// Mitsubishi GX Works2 project: GROUP34   PLC: FX3G

// global labels: Global1
VAR_GLOBAL
  Start_day_button AT X007 : BOOL;
  Insert_stock_once AT M9 : BOOL;
  Petel_input AT D1100 : REAL;
  Petel_stock AT D1102 : REAL;
  Lemon_input AT D1104 : REAL;
  Lemon_stock AT D1106 : REAL;
  Stabilizer_input AT D1108 : REAL;
  Stabilizer_stock AT D1110 : REAL;
  Gummy_input AT D1112 : REAL;
  Gummy_stock AT D1114 : REAL;
  Out_of_stock_reg AT M13 : BOOL;
  Emergency_button AT X005 : BOOL;
  End_day AT M1 : BOOL;
  Start_production AT M2 : BOOL;
  Start_packing AT X004 : BOOL;
  Choose_type AT X001 : BOOL;
END_VAR
VAR_GLOBAL CONSTANT
  Min_petel : REAL := 280;
  Min_lemon : REAL := 455;
  Min_stabilazer : REAL := 105;
  Min_gummy : REAL := 28;
  Min_petel_pinuk : REAL := 385;
  Min_lemon_pinuk : REAL := 665;
  Min_stabilazer_pinuk : REAL := 210;
  Min_gummy_pinuk : REAL := 70;
END_VAR
VAR_GLOBAL
  Out_of_stock_pinuk AT M14 : BOOL;
  Start_day_bulb AT Y007 : BOOL;
  Analog_output AT D8282 : INT;
  Tot_storage AT D1128 : REAL;
END_VAR
VAR_GLOBAL CONSTANT
  Div_analog1 : REAL := 400;
END_VAR
VAR_GLOBAL
  Start_preperation AT M6 : BOOL;
END_VAR
VAR_GLOBAL CONSTANT
  Choose_reg : REAL := 5;
END_VAR
VAR_GLOBAL
  Make_reg AT M7 : BOOL;
  Make_pinuk AT M8 : BOOL;
  Div_output AT D1170 : REAL;
  Is_mix AT TC1 : BOOL;
END_VAR
VAR_GLOBAL CONSTANT
  Wait_5_sec : INT := 50;
END_VAR
VAR_GLOBAL
  Preperation_lamp AT Y000 : BOOL;
  Ice_cream_reg_stage AT M17 : BOOL;
  Ice_cream_pinuk_stage AT M18 : BOOL;
  Petel_preperation AT D1118 : REAL;
END_VAR
VAR_GLOBAL CONSTANT
  Weight_reg_petel_ice_cream : REAL := 350;
END_VAR
VAR_GLOBAL
  Lemon_preperation AT D1120 : REAL;
END_VAR
VAR_GLOBAL CONSTANT
  Weight_reg_lemon_ice_cream : REAL := 490;
  Weight_pinuk_petel_ice_cream : REAL := 560;
  Weight_pinuk_lemon_ice_cream : REAL := 700;
END_VAR
VAR_GLOBAL
  Start_cooling AT X002 : BOOL;
  Cool_petel AT D1122 : REAL;
  Cooling AT M22 : BOOL;
  Is_cooling AT TC2 : BOOL;
END_VAR
VAR_GLOBAL CONSTANT
  Cooling_time : INT := 80;
END_VAR
VAR_GLOBAL
  Cooling_lamp AT M26 : BOOL;
  Temp_sensor_upper10 AT X003 : BOOL;
  Finish_mix AT TS1 : BOOL;
  Finish_cooling AT TS2 : BOOL;
  Cooling_finish AT TS2 : BOOL;
  Cooling_inprocess AT M21 : BOOL;
  Temp_under10 AT M23 : BOOL;
  Cool_lemon AT D1124 : REAL;
  Mix_Tot AT D1126 : REAL;
  Finish_move_icecream AT M25 : BOOL;
END_VAR
VAR_GLOBAL CONSTANT
  Gummy_reg : REAL := 28;
END_VAR
VAR_GLOBAL
  Finish_move AT M24 : BOOL;
END_VAR
VAR_GLOBAL CONSTANT
  Gummy_pinuk : REAL := 70;
END_VAR
VAR_GLOBAL
  Finish_mix_pinuk AT M12 : BOOL;
  Help_Blinking AT M0 : BOOL;
  Blink_y5 AT TC3 : BOOL;
END_VAR
VAR_GLOBAL CONSTANT
  Counter_blink_y5 : INT := 5;
END_VAR
VAR_GLOBAL
  Stop_blink_y5 AT TS3 : BOOL;
  Y5_bulb AT Y005 : BOOL;
  Finish_mix_reg AT M11 : BOOL;
  Blink_y6 AT TC4 : BOOL;
END_VAR
VAR_GLOBAL CONSTANT
  Counter_blink_y6 : INT := 5;
END_VAR
VAR_GLOBAL
  Stop_blink_y6 AT TS4 : BOOL;
  Y6_bulb AT Y006 : BOOL;
  Timer_blinking_reg AT TC5 : BOOL;
END_VAR
VAR_GLOBAL CONSTANT
  Counter_3sec : INT := 30;
END_VAR
VAR_GLOBAL
  Stop_reg_mix AT TS5 : BOOL;
  Timer_blinking_pinuk AT TC6 : BOOL;
END_VAR
VAR_GLOBAL CONSTANT
  Counter_5sec : INT := 50;
END_VAR
VAR_GLOBAL
  Stop_pinuk_mix AT TS6 : BOOL;
  Save_type AT D1200 : REAL;
  Test AT D1500 : REAL;
  Analog_to_real AT D6000 : REAL;
  Insert_to_storage AT X000 : BOOL;
END_VAR
VAR_GLOBAL CONSTANT
  Counter_7 : INT := 7;
END_VAR
VAR_GLOBAL
  Count_in_storage AT CC1 : BOOL;
  Stocking_bulb AT M27 : BOOL;
  finish_stocking AT CS1 : BOOL;
END_VAR
VAR_GLOBAL CONSTANT
  Add_1 : REAL := 1.0;
  Div_analog2 : REAL := 40.0;
END_VAR
VAR_GLOBAL
  num_of_packs AT D1130 : REAL;
  Analog_input1 AT D8280 : INT;
  Cooling_stocking_lamp AT Y002 : BOOL;
  Is_out_of_stock AT M29 : BOOL;
  Finish_cool AT M26 : BOOL;
END_VAR

// task Task_01 (event TRUE, interval 0, priority 31): POU_01

PROGRAM POU_01
(* structured ladder/FBD written out as ST: instructions are called as NAME(EN, inputs, outputs); _pN, _eN, _tN stand for wires *)
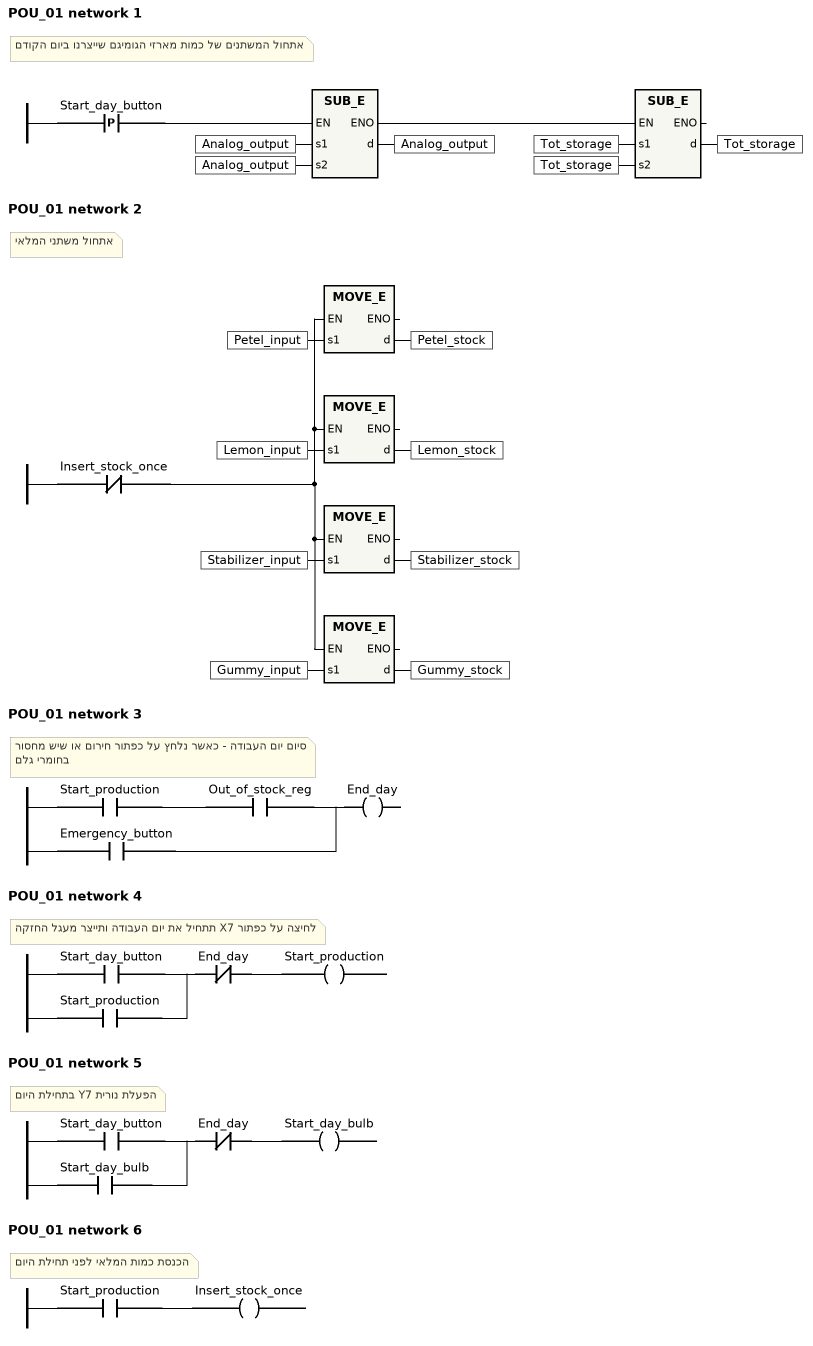
(* network 1 *)
(* אתחול המשתנים של כמות מארזי הגומיגם שייצרנו ביום הקודם *)
_e1 := SUB_E(LDP(TRUE, Start_day_button), Analog_output, Analog_output, Analog_output);
SUB_E(_e1, Tot_storage, Tot_storage, Tot_storage);
(* network 2 *)
(* אתחול משתני המלאי *)
_p1 := NOT Insert_stock_once;
MOVE_E(_p1, Petel_input, Petel_stock);
MOVE_E(_p1, Lemon_input, Lemon_stock);
MOVE_E(_p1, Stabilizer_input, Stabilizer_stock);
MOVE_E(_p1, Gummy_input, Gummy_stock);
(* network 3 *)
(* סיום יום העבודה - כאשר נלחץ על כפתור חירום או שיש מחסור בחומרי גלם *)
End_day := (Start_production AND Out_of_stock_reg) OR Emergency_button;
(* network 4 *)
(* לחיצה על כפתור X7 תתחיל את יום העבודה ותייצר מעגל החזקה *)
Start_production := (Start_day_button OR Start_production) AND NOT End_day;
(* network 5 *)
(* הפעלת נורית Y7 בתחילת היום *)
Start_day_bulb := (Start_day_button OR Start_day_bulb) AND NOT End_day;
(* network 6 *)
(* הכנסת כמות המלאי לפני תחילת היום *)
Insert_stock_once := Start_production;
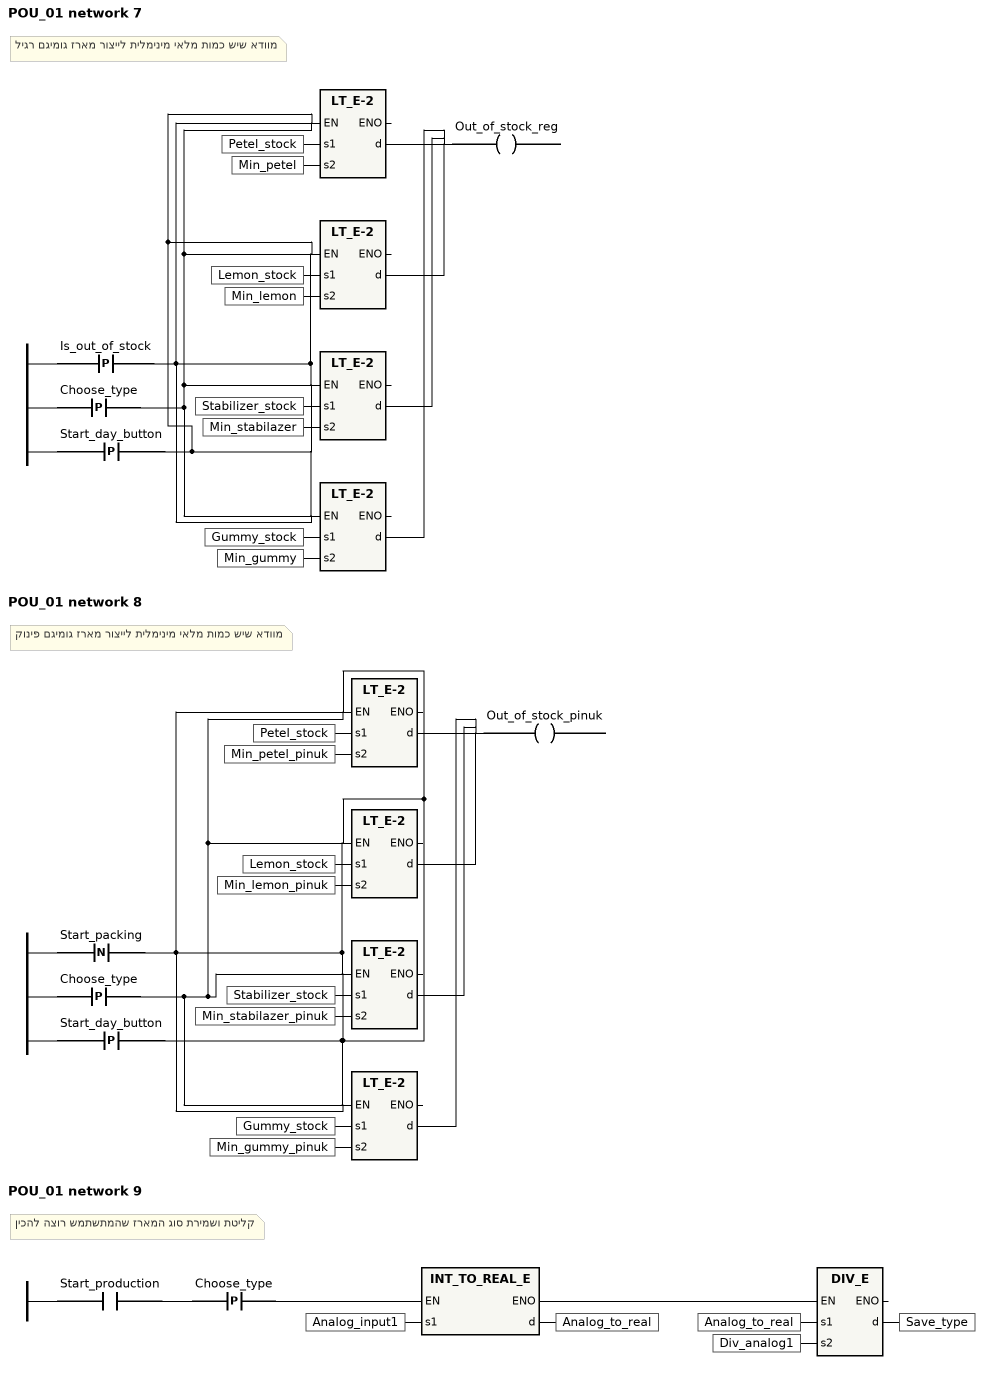
(* network 7 *)
(* מוודא שיש כמות מלאי מינימלית לייצור מארז גומיגם רגיל *)
_p1 := LDP(TRUE, Is_out_of_stock) OR LDP(TRUE, Choose_type) OR LDP(TRUE, Start_day_button);
LT_E(_p1, Petel_stock, Min_petel, _t2);
LT_E(_p1, Lemon_stock, Min_lemon, _t3);
LT_E(_p1, Stabilizer_stock, Min_stabilazer, _t4);
LT_E(_p1, Gummy_stock, Min_gummy, _t5);
Out_of_stock_reg := _t2 OR _t3 OR _t4 OR _t5;
(* network 8 *)
(* מוודא שיש כמות מלאי מינימלית לייצור מארז גומיגם פינוק *)
_p1 := LDF(TRUE, Start_packing) OR LDP(TRUE, Choose_type) OR LDP(TRUE, Start_day_button);
LT_E(_p1, Petel_stock, Min_petel_pinuk, _t2);
LT_E(_p1, Lemon_stock, Min_lemon_pinuk, _t3);
LT_E(_p1, Stabilizer_stock, Min_stabilazer_pinuk, _t4);
LT_E(_p1, Gummy_stock, Min_gummy_pinuk, _t5);
Out_of_stock_pinuk := _t2 OR _t3 OR _t4 OR _t5;
(* network 9 *)
(* קליטת ושמירת סוג המארז שהמתשתמש רוצה להכין *)
_e1 := INT_TO_REAL_E(Start_production AND LDP(TRUE, Choose_type), Analog_input1, Analog_to_real);
DIV_E(_e1, Analog_to_real, Div_analog1, Save_type);
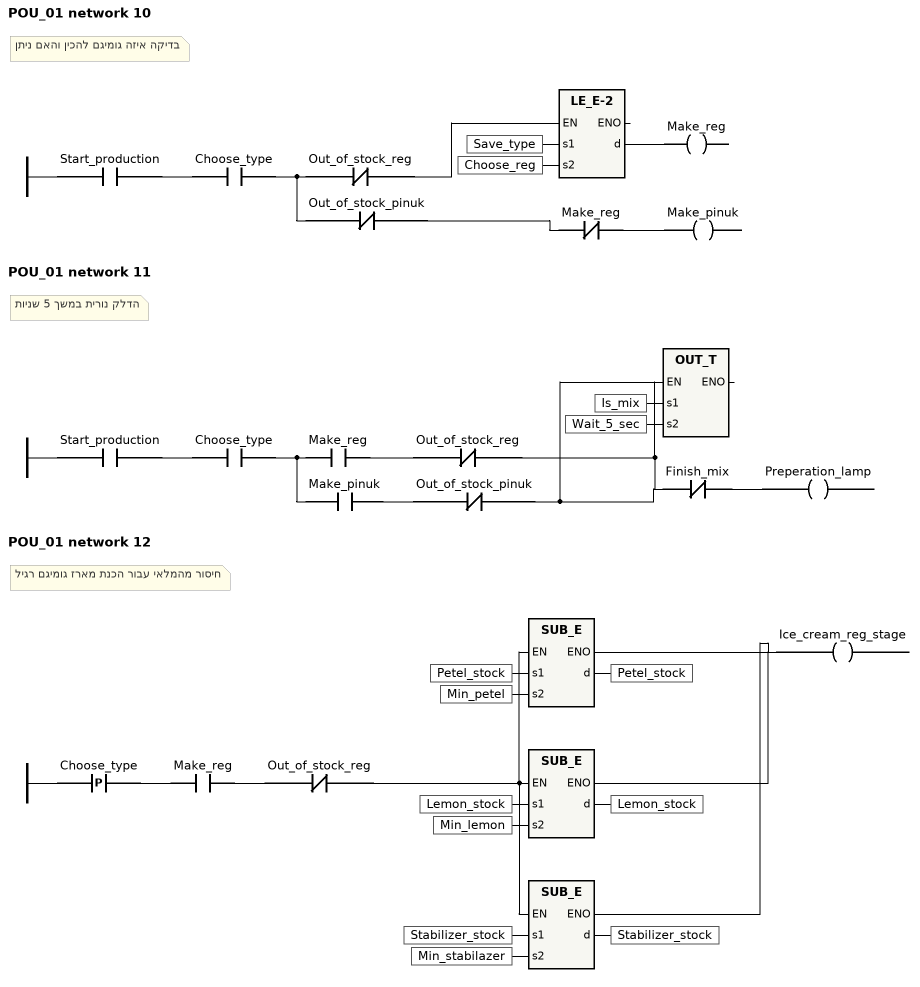
(* network 10 *)
(* בדיקה איזה גומיגם להכין והאם ניתן *)
_p1 := Start_production AND Choose_type;
LE_E(_p1 AND NOT Out_of_stock_reg, Save_type, Choose_reg, _t2);
Make_reg := _t2;
Make_pinuk := _p1 AND NOT Out_of_stock_pinuk AND NOT Make_reg;
(* network 11 *)
(* הדלק נורית במשך 5 שניות *)
_p1 := Start_production AND Choose_type;
_p2 := (_p1 AND Make_reg AND NOT Out_of_stock_reg) OR (_p1 AND Make_pinuk AND NOT Out_of_stock_pinuk);
OUT_T(_p2, Is_mix, Wait_5_sec);
Preperation_lamp := _p2 AND NOT Finish_mix;
(* network 12 *)
(* חיסור מהמלאי עבור הכנת מארז גומיגם רגיל *)
_p1 := LDP(TRUE, Choose_type) AND Make_reg AND NOT Out_of_stock_reg;
_e2 := SUB_E(_p1, Petel_stock, Min_petel, Petel_stock);
_e3 := SUB_E(_p1, Lemon_stock, Min_lemon, Lemon_stock);
_e4 := SUB_E(_p1, Stabilizer_stock, Min_stabilazer, Stabilizer_stock);
Ice_cream_reg_stage := _e2 OR _e3 OR _e4;
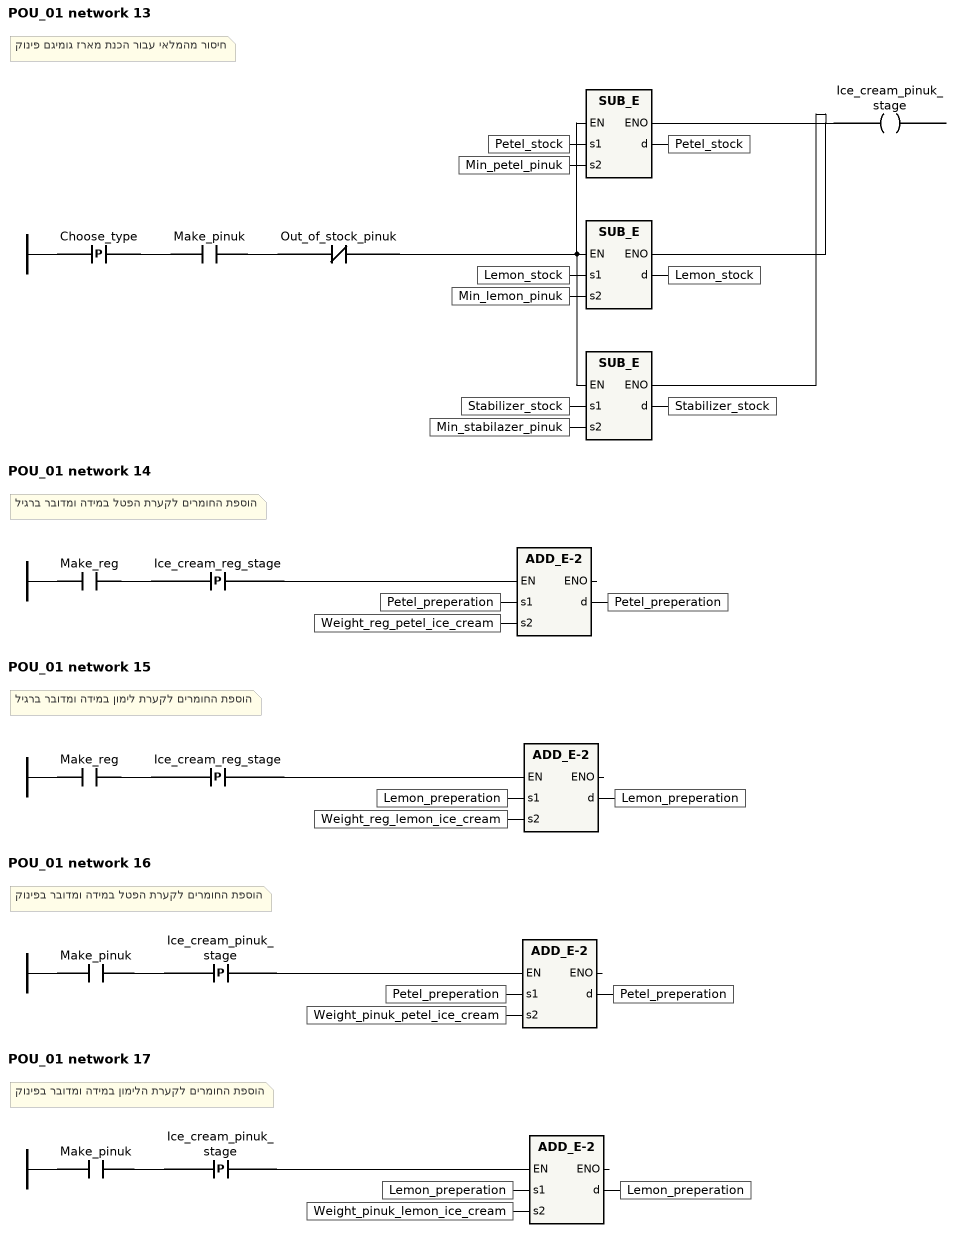
(* network 13 *)
(* חיסור מהמלאי עבור הכנת מארז גומיגם פינוק *)
_p1 := LDP(TRUE, Choose_type) AND Make_pinuk AND NOT Out_of_stock_pinuk;
_e2 := SUB_E(_p1, Petel_stock, Min_petel_pinuk, Petel_stock);
_e3 := SUB_E(_p1, Lemon_stock, Min_lemon_pinuk, Lemon_stock);
_e4 := SUB_E(_p1, Stabilizer_stock, Min_stabilazer_pinuk, Stabilizer_stock);
Ice_cream_pinuk_stage := _e2 OR _e3 OR _e4;
(* network 14 *)
(* הוספת החומרים לקערת הפטל במידה ומדובר ברגיל *)
ADD_E(Make_reg AND LDP(TRUE, Ice_cream_reg_stage), Petel_preperation, Weight_reg_petel_ice_cream, Petel_preperation);
(* network 15 *)
(* הוספת החומרים לקערת לימון במידה ומדובר ברגיל *)
ADD_E(Make_reg AND LDP(TRUE, Ice_cream_reg_stage), Lemon_preperation, Weight_reg_lemon_ice_cream, Lemon_preperation);
(* network 16 *)
(* הוספת החומרים לקערת הפטל במידה ומדובר בפינוק *)
ADD_E(Make_pinuk AND LDP(TRUE, Ice_cream_pinuk_stage), Petel_preperation, Weight_pinuk_petel_ice_cream, Petel_preperation);
(* network 17 *)
(* הוספת החומרים לקערת הלימון במידה ומדובר בפינוק *)
ADD_E(Make_pinuk AND LDP(TRUE, Ice_cream_pinuk_stage), Lemon_preperation, Weight_pinuk_lemon_ice_cream, Lemon_preperation);
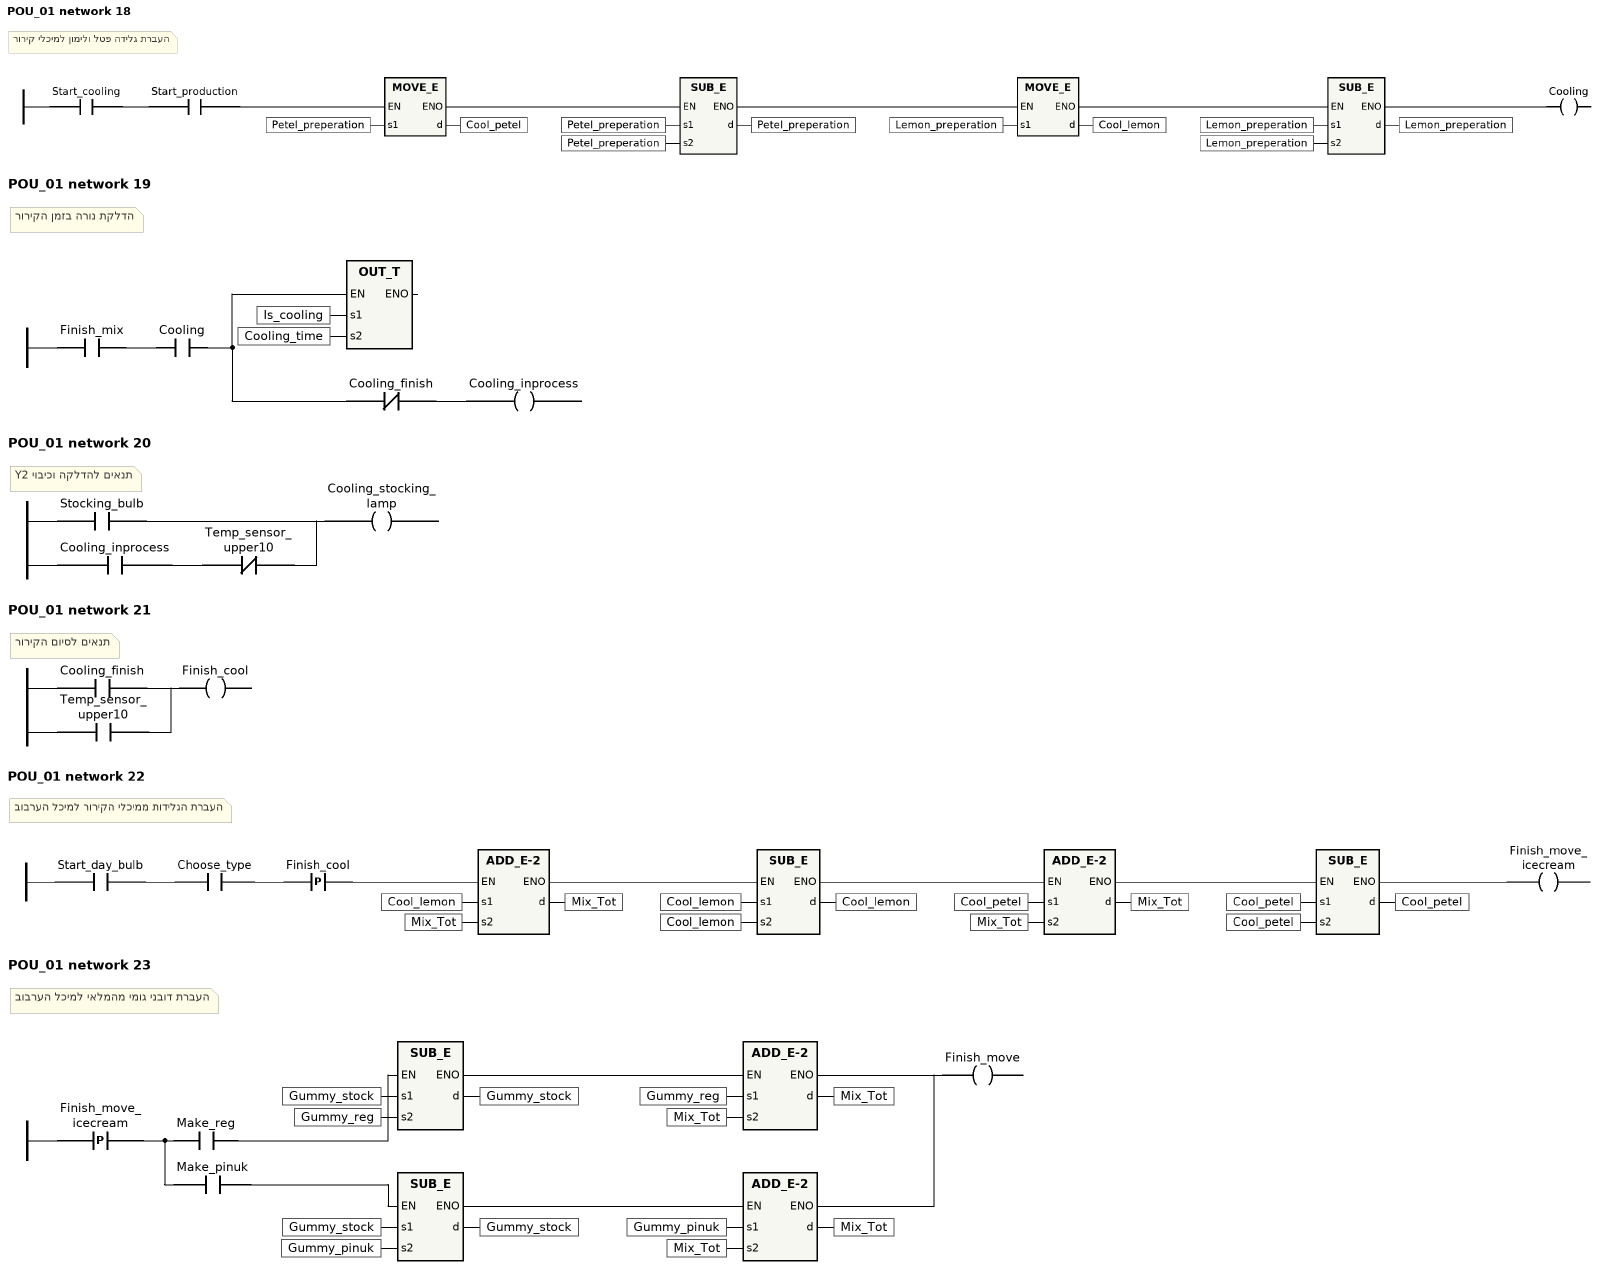
(* network 18 *)
(* העברת גלידה פטל ולימון למיכלי קירור *)
_e1 := MOVE_E(Start_cooling AND Start_production, Petel_preperation, Cool_petel);
_e2 := SUB_E(_e1, Petel_preperation, Petel_preperation, Petel_preperation);
_e3 := MOVE_E(_e2, Lemon_preperation, Cool_lemon);
_e4 := SUB_E(_e3, Lemon_preperation, Lemon_preperation, Lemon_preperation);
Cooling := _e4;
(* network 19 *)
(* הדלקת נורה בזמן הקירור *)
_p1 := Finish_mix AND Cooling;
OUT_T(_p1, Is_cooling, Cooling_time);
Cooling_inprocess := _p1 AND NOT Cooling_finish;
(* network 20 *)
(* תנאים להדלקה וכיבוי Y2 *)
Cooling_stocking_lamp := Stocking_bulb OR (Cooling_inprocess AND NOT Temp_sensor_upper10);
(* network 21 *)
(* תנאים לסיום הקירור *)
Finish_cool := Cooling_finish OR Temp_sensor_upper10;
(* network 22 *)
(* העברת הגלידות ממיכלי הקירור למיכל הערבוב *)
_e1 := ADD_E(Start_day_bulb AND Choose_type AND LDP(TRUE, Finish_cool), Cool_lemon, Mix_Tot, Mix_Tot);
_e2 := SUB_E(_e1, Cool_lemon, Cool_lemon, Cool_lemon);
_e3 := ADD_E(_e2, Cool_petel, Mix_Tot, Mix_Tot);
_e4 := SUB_E(_e3, Cool_petel, Cool_petel, Cool_petel);
Finish_move_icecream := _e4;
(* network 23 *)
(* העברת דובני גומי מהמלאי למיכל הערבוב *)
_p1 := LDP(TRUE, Finish_move_icecream);
_e2 := SUB_E(_p1 AND Make_reg, Gummy_stock, Gummy_reg, Gummy_stock);
_e3 := ADD_E(_e2, Gummy_reg, Mix_Tot, Mix_Tot);
_e4 := SUB_E(_p1 AND Make_pinuk, Gummy_stock, Gummy_pinuk, Gummy_stock);
_e5 := ADD_E(_e4, Gummy_pinuk, Mix_Tot, Mix_Tot);
Finish_move := _e3 OR _e5;
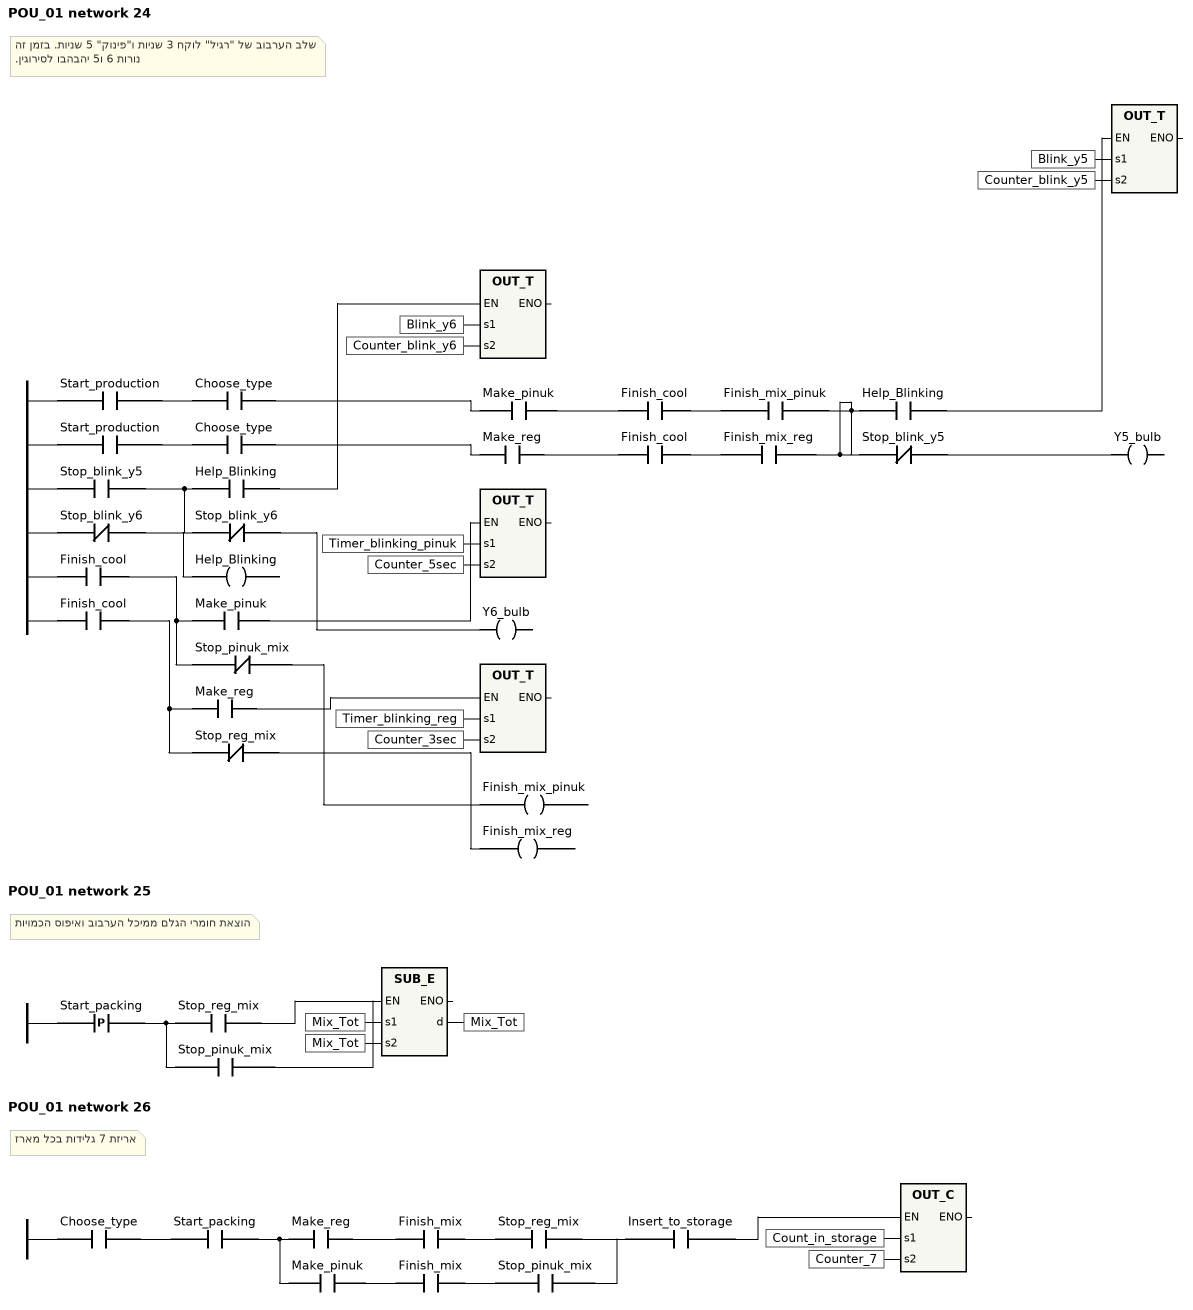
(* network 24 *)
(* שלב הערבוב של "רגיל" לוקח 3 שניות ו"פינוק" 5 שניות. בזמן זה נורות 6 ו5 יהבהבו לסירוגין. *)
_p1 := (Start_production AND Choose_type AND Make_pinuk AND Finish_cool AND Finish_mix_pinuk) OR (Start_production AND Choose_type AND Make_reg AND Finish_cool AND Finish_mix_reg);
OUT_T(_p1 AND Help_Blinking, Blink_y5, Counter_blink_y5);
Y5_bulb := _p1 AND NOT Stop_blink_y5;
OUT_T(Stop_blink_y5 AND Help_Blinking, Blink_y6, Counter_blink_y6);
Y6_bulb := Stop_blink_y5 AND NOT Stop_blink_y6;
Help_Blinking := NOT Stop_blink_y6;
OUT_T(Finish_cool AND Make_pinuk, Timer_blinking_pinuk, Counter_5sec);
Finish_mix_pinuk := Finish_cool AND NOT Stop_pinuk_mix;
OUT_T(Finish_cool AND Make_reg, Timer_blinking_reg, Counter_3sec);
Finish_mix_reg := Finish_cool AND NOT Stop_reg_mix;
(* network 25 *)
(* הוצאת חומרי הגלם ממיכל הערבוב ואיפוס הכמויות *)
_p1 := LDP(TRUE, Start_packing);
SUB_E((_p1 AND Stop_reg_mix) OR (_p1 AND Stop_pinuk_mix), Mix_Tot, Mix_Tot, Mix_Tot);
(* network 26 *)
(* אריזת 7 גלידות בכל מארז *)
_p1 := Choose_type AND Start_packing;
OUT_C(((_p1 AND Make_reg AND Finish_mix AND Stop_reg_mix) OR (_p1 AND Make_pinuk AND Finish_mix AND Stop_pinuk_mix)) AND Insert_to_storage, Count_in_storage, Counter_7);
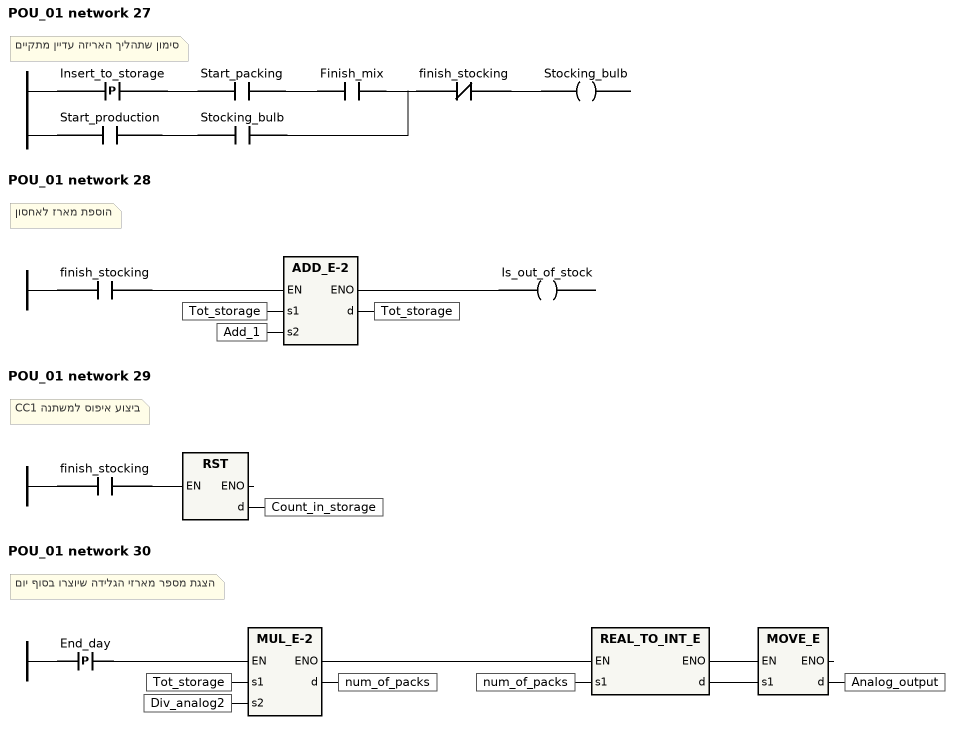
(* network 27 *)
(* סימון שתהליך האריזה עדיין מתקיים *)
Stocking_bulb := ((LDP(TRUE, Insert_to_storage) AND Start_packing AND Finish_mix) OR (Start_production AND Stocking_bulb)) AND NOT finish_stocking;
(* network 28 *)
(* הוספת מארז לאחסון *)
_e1 := ADD_E(finish_stocking, Tot_storage, Add_1, Tot_storage);
Is_out_of_stock := _e1;
(* network 29 *)
(* ביצוע איפוס למשתנה CC1 *)
RST(finish_stocking, Count_in_storage);
(* network 30 *)
(* הצגת מספר מארזי הגלידה שיוצרו בסוף יום *)
_e1 := MUL_E(LDP(TRUE, End_day), Tot_storage, Div_analog2, num_of_packs);
_e3 := REAL_TO_INT_E(_e1, num_of_packs, _t2);
MOVE_E(_e3, _t2, Analog_output);
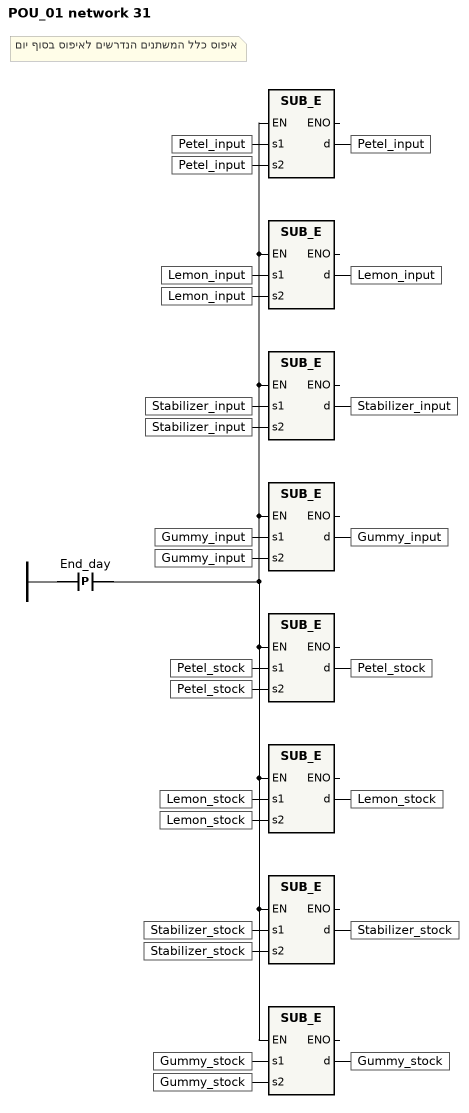
(* network 31 *)
(* איפוס כלל המשתנים הנדרשים לאיפוס בסוף יום *)
_p1 := LDP(TRUE, End_day);
SUB_E(_p1, Petel_input, Petel_input, Petel_input);
SUB_E(_p1, Lemon_input, Lemon_input, Lemon_input);
SUB_E(_p1, Stabilizer_input, Stabilizer_input, Stabilizer_input);
SUB_E(_p1, Gummy_input, Gummy_input, Gummy_input);
SUB_E(_p1, Petel_stock, Petel_stock, Petel_stock);
SUB_E(_p1, Lemon_stock, Lemon_stock, Lemon_stock);
SUB_E(_p1, Stabilizer_stock, Stabilizer_stock, Stabilizer_stock);
SUB_E(_p1, Gummy_stock, Gummy_stock, Gummy_stock);
END_PROGRAM
